// TIA Portal V17 export
// export: Created 2023-12-22T15:05:35.4318091Z, ExportSetting WithDefaults, DisplayName Totally Integrated Automation Portal, DisplayVersion V17, DisplayName TIA Portal Openness, DisplayVersion V17, DisplayName TIA Portal Version Control Interface, DisplayVersion V17, DisplayName STEP 7 Professional, DisplayVersion V17, DisplayName STEP 7 Safety, DisplayVersion V17, DisplayName WinCC Advanced, DisplayVersion V17
TYPE "Line_Report"
// stored: IsFailsafeCompliant false
   STRUCT
      RM_1 : Real;   // Расход без разбавления
      RM_2 : Real;   // Расход с разбавлением
      Res_1 : Real;   // Наработка насоса 1, часы
      Res_2 : Real;   // Наработка насоса 2, часы
      D_Mid : Real;   // Средняя доза за сутки
      Flow : Real;   // Общая труба (куда происходит дозация)
      WeekDay : Int;   // День недели
      Day : Int;   // Дата записи
      Month : Int;   // Месяц записи
   END_STRUCT;
END_TYPE
